FUNCTION_BLOCK Q_CtrlAudioSignal (* Command Control audio device ( Part 6 - F.10 ). *)
  (* Standard: ISO 11783-6; Description: This command can be used to control the audio on the VT. Return values iso_s16 - E_NO_ERR - OK - E_OVERFLOW - buffer overflow - E_NOACT - Command not possible in current state - E_NO_INSTANCE - No VT client available *)
  (* Version 1.0, 2022-07-08, franz *)
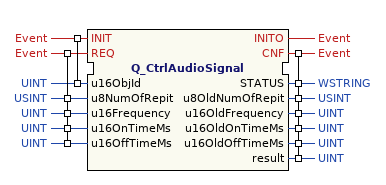
  EVENT_INPUT
    INIT WITH u16ObjId; (* Service Initialization *)
    REQ WITH u8NumOfRepit, u16Frequency, u16OnTimeMs, u16OffTimeMs; (* Service Request *)
  END_EVENT
  EVENT_OUTPUT
    INITO; (* Initialization Confirm *)
    CNF WITH STATUS, u16OldOnTimeMs, u8OldNumOfRepit, u16OldFrequency, result, u16OldOffTimeMs; (* Confirmation of Requested Service *)
  END_EVENT
  VAR_INPUT
    u16ObjId : UINT; (* Object ID *)
    u8NumOfRepit : USINT; (* Number of repetitions Range: 1 - 255 *)
    u16Frequency : UINT; (* Frequency *)
    u16OnTimeMs : UINT; (* On time duration in ms *)
    u16OffTimeMs : UINT; (* Off time duration in ms *)
  END_VAR
  VAR_OUTPUT
    STATUS : WSTRING; (* Service Status *)
    u8OldNumOfRepit : USINT; (* Old Number of repetitions Range: 1 - 255 *)
    u16OldFrequency : UINT; (* Old Frequency *)
    u16OldOnTimeMs : UINT; (* Old on time duration in ms *)
    u16OldOffTimeMs : UINT; (* Old off time duration in ms *)
    result : UINT; (* retval see description *)
  END_VAR
END_FUNCTION_BLOCK
